KUKA KRL program: ps_ltc_res_c2.src, ps_ltc_res_c2.dat

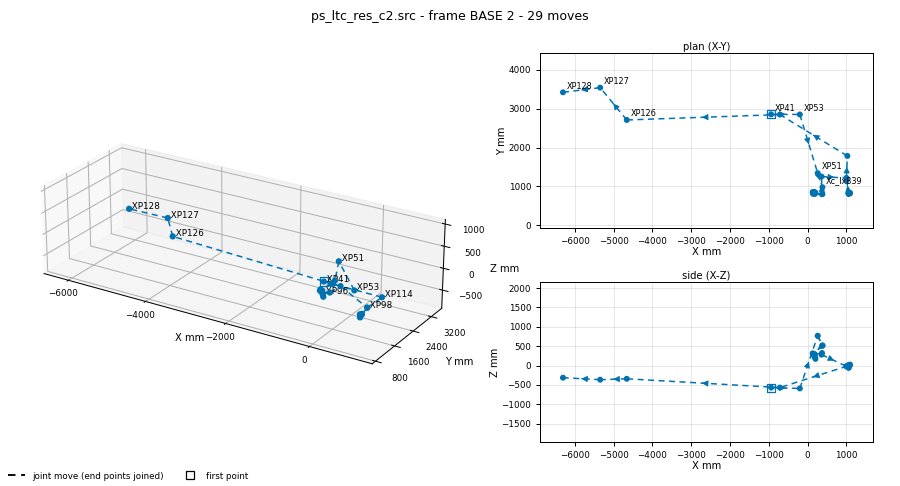
[picture p0: tool path of ps_ltc_res_c2.src in frame BASE 2, 29 of 30 moves have a stored position in this frame; points joined in program order, loops and branches not executed]
--- ps_ltc_res_c2.src ---
&ACCESS RVO2
&REL 51
&COMMENT Solda GUN C2 Respot
&PARAM DISKPATH = KRC:\R1\Program
DEF ps_ltc_res_c2( )
;FOLD INI
;FOLD SPOTTECH INI
USERSPOT(#INIT)
;ENDFOLD (SPOTTECH INI)
  ;FOLD USER INI
    ;Make your modifications here

  ;ENDFOLD (USER INI)
;ENDFOLD (INI)

; Caracterização dos meios de produção:
; Versão Atual:
; 15/07/2013 12:00 Name: P13.050-R4 CHANGES: Respot Acelo
; Pinça C2

chk_w2_wechs_ok ( )     ; CHECK FERRAMENTA: C2

;FOLD PTP P41 CONT Vel=100 % PDAT36 Tool[2]:GUN C2 Base[2]:ACCELO;%{PE}%R 8.2.20,%MKUKATPBASIS,%CMOVE,%VPTP,%P 1:PTP, 2:P41, 3:C_DIS, 5:100, 7:PDAT36
$BWDSTART=FALSE
PDAT_ACT=PPDAT36
FDAT_ACT=FP41
BAS(#PTP_PARAMS,100)
PTP XP41 C_DIS
;ENDFOLD

;FOLD OUT 3334 'R4 liberacao para solda respot' State=TRUE ;%{PE}%R 8.2.20,%MKUKATPBASIS,%COUT,%VOUTX,%P 2:3334, 3:R4 liberacao para solda respot, 5:TRUE, 6:
$OUT[3334]=TRUE
;ENDFOLD
;FOLD WAIT FOR ( IN 3334 'Aguarda lib soldar respot' );%{PE}%R 8.2.20,%MKUKATPBASIS,%CEXT_WAIT_FOR,%VEXT_WAIT_FOR,%P 2:, 4:, 5:$IN, 6:3334, 7:Aguarda lib soldar respot, 9:
WAIT FOR  ( $IN[3334] )
;ENDFOLD
;FOLD OUT 3334 'R4 solda respot concluida' State=FALSE ;%{PE}%R 8.2.20,%MKUKATPBASIS,%COUT,%VOUTX,%P 2:3334, 3:R4 solda respot concluida, 5:FALSE, 6:
$OUT[3334]=FALSE
;ENDFOLD
;FOLD OUT 3348 'Fora area GEOBOX' State=FALSE ;%{PE}%R 8.2.20,%MKUKATPBASIS,%COUT,%VOUTX,%P 2:3348, 3:Fora area GEOBOX, 5:FALSE, 6:
$OUT[3348]=FALSE
;ENDFOLD

;FOLD PTP P53 CONT Vel=100 % PDAT53 Tool[2]:GUN C2 Base[2]:ACCELO;%{PE}%R 8.2.20,%MKUKATPBASIS,%CMOVE,%VPTP,%P 1:PTP, 2:P53, 3:C_DIS, 5:100, 7:PDAT53
$BWDSTART=FALSE
PDAT_ACT=PPDAT53
FDAT_ACT=FP53
BAS(#PTP_PARAMS,100)
PTP XP53 C_DIS
;ENDFOLD
;FOLD PTP P51 CONT Vel=100 % PDAT51 Tool[2]:GUN C2 Base[2]:ACCELO;%{PE}%R 8.2.20,%MKUKATPBASIS,%CMOVE,%VPTP,%P 1:PTP, 2:P51, 3:C_DIS, 5:100, 7:PDAT51
$BWDSTART=FALSE
PDAT_ACT=PPDAT51
FDAT_ACT=FP51
BAS(#PTP_PARAMS,100)
PTP XP51 C_DIS
;ENDFOLD
;FOLD PTP c_lx839 CONT Vel=100 % P_OLP118 Tool[2]:GUN C2 Base[2]:ACCELO;%{PE}%R 8.2.20,%MKUKATPBASIS,%CMOVE,%VPTP,%P 1:PTP, 2:c_lx839, 3:C_DIS, 5:100, 7:P_OLP118
$BWDSTART=FALSE
PDAT_ACT=PP_OLP118
FDAT_ACT=Fc_lx839
BAS(#PTP_PARAMS,100)
PTP Xc_lx839 C_DIS
;ENDFOLD
;FOLD PTP P95 CONT Vel=100 % PDAT110 Tool[2]:GUN C2 Base[2]:ACCELO;%{PE}%R 8.2.20,%MKUKATPBASIS,%CMOVE,%VPTP,%P 1:PTP, 2:P95, 3:C_DIS, 5:100, 7:PDAT110
$BWDSTART=FALSE
PDAT_ACT=PPDAT110
FDAT_ACT=FP95
BAS(#PTP_PARAMS,100)
PTP XP95 C_DIS
;ENDFOLD
;FOLD PTP c_lx840 CONT Vel=100 % P_OLP119 Tool[2]:GUN C2 Base[2]:ACCELO;%{PE}%R 8.2.20,%MKUKATPBASIS,%CMOVE,%VPTP,%P 1:PTP, 2:c_lx840, 3:C_DIS, 5:100, 7:P_OLP119
$BWDSTART=FALSE
PDAT_ACT=PP_OLP119
FDAT_ACT=Fc_lx840
BAS(#PTP_PARAMS,100)
PTP Xc_lx840 C_DIS
;ENDFOLD

;FOLD ; swp_60_0224;%{PE}%R 8.2.20,%MKUKATPBASIS,%CCOMMENT,%VNORMAL,%P 2:swp_60_0224
;ENDFOLD
;FOLD PTP swp_60_0224 P_OLP120 SPOT Gun=2 RETR CLS PGNO1=106 ACTIVE=1 Tool[2]:GUN C2 Base[2]:ACCELO;%{PE}%R 8.2.2,%MKUKATPSPOT,%CSPOT,%VPTP,%P 1:PTP, 2:swp_60_0224, 3:, 5:100, 7:P_OLP120, 10:2, 12:#FIRST, 14:#CLO, 16:147, 18:1, 20:1, 22:0, 24:1, 25:S_OLP6
$BWDSTART=FALSE
PDAT_ACT=PP_OLP120
FDAT_ACT=Fswp_60_0224
BAS(#PTP_PARAMS,PP_OLP120.VEL)
S_ACT.GUN=2
S_ACT.PAIR=SDEFAULT.PAIR
S_ACT.RETR=#CLO
S_ACT.CLO_TM=1
S_ACT.PGNO1=106
S_ACT.PGNO2=SDEFAULT.PGNO2
S_ACT.PRESS1=SDEFAULT.PRESS1
S_ACT.PRESS2=SDEFAULT.PRESS2
S_READY=FALSE
PTP Xswp_60_0224
USERSPOT(#SPOT, S_ACT)
WAIT FOR S_READY
;ENDFOLD

;FOLD PTP c_lx841 CONT Vel=100 % P_OLP121 Tool[2]:GUN C2 Base[0];%{PE}%R 8.2.20,%MKUKATPBASIS,%CMOVE,%VPTP,%P 1:PTP, 2:c_lx841, 3:C_DIS, 5:100, 7:P_OLP121
$BWDSTART=FALSE
PDAT_ACT=PP_OLP121
FDAT_ACT=Fc_lx841
BAS(#PTP_PARAMS,100)
PTP Xc_lx841 C_DIS
;ENDFOLD

;FOLD ; swp_60_0228;%{PE}%R 8.2.20,%MKUKATPBASIS,%CCOMMENT,%VNORMAL,%P 2:swp_60_0228
;ENDFOLD
;FOLD PTP swp_60_0228 P_OLP122 SPOT Gun=2 RETR CLS PGNO1=138 ACTIVE=1 Tool[2]:GUN C2 Base[2]:ACCELO;%{PE}%R 8.2.2,%MKUKATPSPOT,%CSPOT,%VPTP,%P 1:PTP, 2:swp_60_0228, 3:, 5:100, 7:P_OLP122, 10:2, 12:#FIRST, 14:#CLO, 16:179, 18:1, 20:1, 22:0, 24:1, 25:S_OLP7
$BWDSTART=FALSE
PDAT_ACT=PP_OLP122
FDAT_ACT=Fswp_60_0228
BAS(#PTP_PARAMS,PP_OLP122.VEL)
S_ACT.GUN=2
S_ACT.PAIR=SDEFAULT.PAIR
S_ACT.RETR=#CLO
S_ACT.CLO_TM=1
S_ACT.PGNO1=138
S_ACT.PGNO2=SDEFAULT.PGNO2
S_ACT.PRESS1=SDEFAULT.PRESS1
S_ACT.PRESS2=SDEFAULT.PRESS2
S_READY=FALSE
PTP Xswp_60_0228
USERSPOT(#SPOT, S_ACT)
WAIT FOR S_READY
;ENDFOLD

;FOLD ; swp_60_0232;%{PE}%R 8.2.20,%MKUKATPBASIS,%CCOMMENT,%VNORMAL,%P 2:swp_60_0232
;ENDFOLD
;FOLD PTP swp_60_0232 P_OLP123 SPOT Gun=2 RETR CLS PGNO1=104 ACTIVE=1 Tool[2]:GUN C2 Base[2]:ACCELO;%{PE}%R 8.2.2,%MKUKATPSPOT,%CSPOT,%VPTP,%P 1:PTP, 2:swp_60_0232, 3:, 5:100, 7:P_OLP123, 10:2, 12:#FIRST, 14:#CLO, 16:145, 18:1, 20:1, 22:0, 24:1, 25:S_OLP8
$BWDSTART=FALSE
PDAT_ACT=PP_OLP123
FDAT_ACT=Fswp_60_0232
BAS(#PTP_PARAMS,PP_OLP123.VEL)
S_ACT.GUN=2
S_ACT.PAIR=SDEFAULT.PAIR
S_ACT.RETR=#CLO
S_ACT.CLO_TM=1
S_ACT.PGNO1=104
S_ACT.PGNO2=SDEFAULT.PGNO2
S_ACT.PRESS1=SDEFAULT.PRESS1
S_ACT.PRESS2=SDEFAULT.PRESS2
S_READY=FALSE
PTP Xswp_60_0232
USERSPOT(#SPOT, S_ACT)
WAIT FOR S_READY
;ENDFOLD

;FOLD PTP P96 CONT Vel=100 % PDAT111 Tool[2]:GUN C2 Base[2]:ACCELO;%{PE}%R 8.2.20,%MKUKATPBASIS,%CMOVE,%VPTP,%P 1:PTP, 2:P96, 3:C_DIS, 5:100, 7:PDAT111
$BWDSTART=FALSE
PDAT_ACT=PPDAT111
FDAT_ACT=FP96
BAS(#PTP_PARAMS,100)
PTP XP96 C_DIS
;ENDFOLD

;FOLD ; swp_60_0234;%{PE}%R 8.2.20,%MKUKATPBASIS,%CCOMMENT,%VNORMAL,%P 2:swp_60_0234
;ENDFOLD
;FOLD PTP swp_60_0234 PDAT112 SPOT Gun=2 RETR OPN PGNO1=103 ACTIVE=1 Tool[2]:GUN C2 Base[2]:ACCELO;%{PE}%R 8.2.2,%MKUKATPSPOT,%CSPOT,%VPTP,%P 1:PTP, 2:swp_60_0234, 3:, 5:100, 7:PDAT112, 10:2, 12:#FIRST, 14:#OPN, 16:144, 18:1, 20:0, 22:0, 24:1, 25:NORMAL
$BWDSTART=FALSE
PDAT_ACT=PPDAT112
FDAT_ACT=Fswp_60_0234
BAS(#PTP_PARAMS,PPDAT112.VEL)
S_ACT.GUN=2
S_ACT.PAIR=SDEFAULT.PAIR
S_ACT.RETR=#OPN
S_ACT.CLO_TM=1
S_ACT.PGNO1=103
S_ACT.PGNO2=SDEFAULT.PGNO2
S_ACT.PRESS1=SDEFAULT.PRESS1
S_ACT.PRESS2=SDEFAULT.PRESS2
S_READY=FALSE
PTP Xswp_60_0234
USERSPOT(#SPOT, S_ACT)
WAIT FOR S_READY
;ENDFOLD

;FOLD PTP c_lx804 CONT Vel=100 % P_OLP124 Tool[2]:GUN C2 Base[2]:ACCELO;%{PE}%R 8.2.20,%MKUKATPBASIS,%CMOVE,%VPTP,%P 1:PTP, 2:c_lx804, 3:C_DIS, 5:100, 7:P_OLP124
$BWDSTART=FALSE
PDAT_ACT=PP_OLP124
FDAT_ACT=Fc_lx804
BAS(#PTP_PARAMS,100)
PTP Xc_lx804 C_DIS
;ENDFOLD
;FOLD PTP P94 CONT Vel=100 % PDAT109 Tool[2]:GUN C2 Base[2]:ACCELO;%{PE}%R 8.2.20,%MKUKATPBASIS,%CMOVE,%VPTP,%P 1:PTP, 2:P94, 3:C_DIS, 5:100, 7:PDAT109
$BWDSTART=FALSE
PDAT_ACT=PPDAT109
FDAT_ACT=FP94
BAS(#PTP_PARAMS,100)
PTP XP94 C_DIS
;ENDFOLD
;FOLD PTP c_lx807 Vel=100 % P_OLP125 Tool[2]:GUN C2 Base[2]:ACCELO;%{PE}%R 8.2.20,%MKUKATPBASIS,%CMOVE,%VPTP,%P 1:PTP, 2:c_lx807, 3:, 5:100, 7:P_OLP125
$BWDSTART=FALSE
PDAT_ACT=PP_OLP125
FDAT_ACT=Fc_lx807
BAS(#PTP_PARAMS,100)
PTP Xc_lx807
;ENDFOLD

;FOLD Collision.Monitoring_AREA_1_On ;%{PE}%MKUKATPUSER
COLLSTOP( 7, 1 ) ;not Interrupt-Controlled
;ENDFOLD

;FOLD PTP P98 CONT Vel=100 % PDAT114 Tool[2]:GUN C2 Base[2]:ACCELO;%{PE}%R 8.2.20,%MKUKATPBASIS,%CMOVE,%VPTP,%P 1:PTP, 2:P98, 3:C_DIS, 5:100, 7:PDAT114
$BWDSTART=FALSE
PDAT_ACT=PPDAT114
FDAT_ACT=FP98
BAS(#PTP_PARAMS,100)
PTP XP98 C_DIS
;ENDFOLD
;FOLD PTP P99 CONT Vel=100 % PDAT115 Tool[2]:GUN C2 Base[2]:ACCELO;%{PE}%R 8.2.20,%MKUKATPBASIS,%CMOVE,%VPTP,%P 1:PTP, 2:P99, 3:C_DIS, 5:100, 7:PDAT115
$BWDSTART=FALSE
PDAT_ACT=PPDAT115
FDAT_ACT=FP99
BAS(#PTP_PARAMS,100)
PTP XP99 C_DIS
;ENDFOLD
;FOLD PTP P100 CONT Vel=100 % PDAT116 Tool[2]:GUN C2 Base[2]:ACCELO;%{PE}%R 8.2.20,%MKUKATPBASIS,%CMOVE,%VPTP,%P 1:PTP, 2:P100, 3:C_DIS, 5:100, 7:PDAT116
$BWDSTART=FALSE
PDAT_ACT=PPDAT116
FDAT_ACT=FP100
BAS(#PTP_PARAMS,100)
PTP XP100 C_DIS
;ENDFOLD
;FOLD PTP P101 CONT Vel=100 % PDAT118 Tool[2]:GUN C2 Base[2]:ACCELO;%{PE}%R 8.2.20,%MKUKATPBASIS,%CMOVE,%VPTP,%P 1:PTP, 2:P101, 3:C_DIS, 5:100, 7:PDAT118
$BWDSTART=FALSE
PDAT_ACT=PPDAT118
FDAT_ACT=FP101
BAS(#PTP_PARAMS,100)
PTP XP101 C_DIS
;ENDFOLD

;FOLD ; 60_0310;%{PE}%R 8.2.20,%MKUKATPBASIS,%CCOMMENT,%VNORMAL,%P 2:60_0310
;ENDFOLD
;FOLD PTP swp_60_0310 PDAT128 SPOT Gun=2 RETR CLS PGNO1=85 ACTIVE=1 Tool[2]:GUN C2 Base[2]:ACCELO;%{PE}%R 8.2.2,%MKUKATPSPOT,%CSPOT,%VPTP,%P 1:PTP, 2:swp_60_0310, 3:, 5:100, 7:PDAT128, 10:2, 12:#FIRST, 14:#CLO, 16:126, 18:1, 20:0, 22:0, 24:1, 25:NORMAL
$BWDSTART=FALSE
PDAT_ACT=PPDAT128
FDAT_ACT=Fswp_60_0310
BAS(#PTP_PARAMS,PPDAT128.VEL)
S_ACT.GUN=2
S_ACT.PAIR=SDEFAULT.PAIR
S_ACT.RETR=#CLO
S_ACT.CLO_TM=1
S_ACT.PGNO1=85
S_ACT.PGNO2=SDEFAULT.PGNO2
S_ACT.PRESS1=SDEFAULT.PRESS1
S_ACT.PRESS2=SDEFAULT.PRESS2
S_READY=FALSE
PTP Xswp_60_0310
USERSPOT(#SPOT, S_ACT)
WAIT FOR S_READY
;ENDFOLD

;FOLD ; 60_0308;%{PE}%R 8.2.20,%MKUKATPBASIS,%CCOMMENT,%VNORMAL,%P 2:60_0308
;ENDFOLD
;FOLD PTP swp_60_0308 PDAT129 SPOT Gun=2 RETR OPN PGNO1=139 ACTIVE=1 Tool[2]:GUN C2 Base[2]:ACCELO;%{PE}%R 8.2.2,%MKUKATPSPOT,%CSPOT,%VPTP,%P 1:PTP, 2:swp_60_0308, 3:, 5:100, 7:PDAT129, 10:2, 12:#FIRST, 14:#OPN, 16:180, 18:1, 20:0, 22:0, 24:1, 25:NORMAL
$BWDSTART=FALSE
PDAT_ACT=PPDAT129
FDAT_ACT=Fswp_60_0308
BAS(#PTP_PARAMS,PPDAT129.VEL)
S_ACT.GUN=2
S_ACT.PAIR=SDEFAULT.PAIR
S_ACT.RETR=#OPN
S_ACT.CLO_TM=1
S_ACT.PGNO1=139
S_ACT.PGNO2=SDEFAULT.PGNO2
S_ACT.PRESS1=SDEFAULT.PRESS1
S_ACT.PRESS2=SDEFAULT.PRESS2
S_READY=FALSE
PTP Xswp_60_0308
USERSPOT(#SPOT, S_ACT)
WAIT FOR S_READY
;ENDFOLD

;FOLD PTP P110 CONT Vel=100 % PDAT130 Tool[2]:GUN C2 Base[2]:ACCELO;%{PE}%R 8.2.20,%MKUKATPBASIS,%CMOVE,%VPTP,%P 1:PTP, 2:P110, 3:C_DIS, 5:100, 7:PDAT130
$BWDSTART=FALSE
PDAT_ACT=PPDAT130
FDAT_ACT=FP110
BAS(#PTP_PARAMS,100)
PTP XP110 C_DIS
;ENDFOLD
;FOLD PTP P111 CONT Vel=100 % PDAT131 Tool[2]:GUN C2 Base[2]:ACCELO;%{PE}%R 8.2.20,%MKUKATPBASIS,%CMOVE,%VPTP,%P 1:PTP, 2:P111, 3:C_DIS, 5:100, 7:PDAT131
$BWDSTART=FALSE
PDAT_ACT=PPDAT131
FDAT_ACT=FP111
BAS(#PTP_PARAMS,100)
PTP XP111 C_DIS
;ENDFOLD
;FOLD PTP P112 CONT Vel=100 % PDAT132 Tool[2]:GUN C2 Base[2]:ACCELO;%{PE}%R 8.2.20,%MKUKATPBASIS,%CMOVE,%VPTP,%P 1:PTP, 2:P112, 3:C_DIS, 5:100, 7:PDAT132
$BWDSTART=FALSE
PDAT_ACT=PPDAT132
FDAT_ACT=FP112
BAS(#PTP_PARAMS,100)
PTP XP112 C_DIS
;ENDFOLD
;FOLD PTP P114 CONT Vel=100 % PDAT134 Tool[2]:GUN C2 Base[2]:ACCELO;%{PE}%R 8.2.20,%MKUKATPBASIS,%CMOVE,%VPTP,%P 1:PTP, 2:P114, 3:C_DIS, 5:100, 7:PDAT134
$BWDSTART=FALSE
PDAT_ACT=PPDAT134
FDAT_ACT=FP114
BAS(#PTP_PARAMS,100)
PTP XP114 C_DIS
;ENDFOLD
;FOLD PTP P109 CONT Vel=100 % PDAT127 Tool[2]:GUN C2 Base[2]:ACCELO;%{PE}%R 8.2.20,%MKUKATPBASIS,%CMOVE,%VPTP,%P 1:PTP, 2:P109, 3:C_DIS, 5:100, 7:PDAT127
$BWDSTART=FALSE
PDAT_ACT=PPDAT127
FDAT_ACT=FP109
BAS(#PTP_PARAMS,100)
PTP XP109 C_DIS
;ENDFOLD
;FOLD PTP P126 CONT Vel=100 % PDAT146 Tool[2]:GUN C2 Base[2]:ACCELO;%{PE}%R 8.2.20,%MKUKATPBASIS,%CMOVE,%VPTP,%P 1:PTP, 2:P126, 3:C_DIS, 5:100, 7:PDAT146
$BWDSTART=FALSE
PDAT_ACT=PPDAT146
FDAT_ACT=FP126
BAS(#PTP_PARAMS,100)
PTP XP126 C_DIS
;ENDFOLD
;FOLD PTP P127 CONT Vel=100 % PDAT147 Tool[2]:GUN C2 Base[2]:ACCELO;%{PE}%R 8.2.20,%MKUKATPBASIS,%CMOVE,%VPTP,%P 1:PTP, 2:P127, 3:C_DIS, 5:100, 7:PDAT147
$BWDSTART=FALSE
PDAT_ACT=PPDAT147
FDAT_ACT=FP127
BAS(#PTP_PARAMS,100)
PTP XP127 C_DIS
;ENDFOLD
;FOLD PTP P128 CONT Vel=100 % PDAT148 Tool[2]:GUN C2 Base[2]:ACCELO;%{PE}%R 8.2.20,%MKUKATPBASIS,%CMOVE,%VPTP,%P 1:PTP, 2:P128, 3:C_DIS, 5:100, 7:PDAT148
$BWDSTART=FALSE
PDAT_ACT=PPDAT148
FDAT_ACT=FP128
BAS(#PTP_PARAMS,100)
PTP XP128 C_DIS
;ENDFOLD

;FOLD PULSE 3345 'Solda Respot concluida' State=TRUE Time=1 sec;%{PE}%R 8.2.20,%MKUKATPBASIS,%COUT,%VPULSE,%P 2:3345, 3:Solda Respot concluida, 5:TRUE, 6:, 8:1
PULSE($OUT[3345], TRUE,1)
;ENDFOLD
;FOLD OUT 3348 'Fora area GEOBOX' State=TRUE ;%{PE}%R 8.2.20,%MKUKATPBASIS,%COUT,%VOUTX,%P 2:3348, 3:Fora area GEOBOX, 5:TRUE, 6:
$OUT[3348]=TRUE
;ENDFOLD
;FOLD Collision.Monitoring_AREA_1_Off . ;%{PE}%MKUKATPUSER
COLLSTOP( 7, 2+0 )
;ENDFOLD

;FOLD PTP P121 Vel=100 % PDAT141 Tool[2]:GUN C2 Base[0];%{PE}%R 8.2.20,%MKUKATPBASIS,%CMOVE,%VPTP,%P 1:PTP, 2:P121, 3:, 5:100, 7:PDAT141
$BWDSTART=FALSE
PDAT_ACT=PPDAT141
FDAT_ACT=FP121
BAS(#PTP_PARAMS,100)
PTP XP121
;ENDFOLD

if FraesAnf (2) then
  f_fraes2 ()
endif

END

--- ps_ltc_res_c2.dat ---
&ACCESS RVO2
&REL 51
&COMMENT Solda GUN C2 Respot
&PARAM DISKPATH = KRC:\R1\Program
DEFDAT  ps_ltc_res_c2
;FOLD EXTERNAL DECLARATIONS;%{PE}%MKUKATPBASIS,%CEXT,%VCOMMON,%P
;FOLD GRIPPERTECH EXT
EXT  H50 (INT  :IN,INT  :IN,INT  :IN,GRP_TYP  :IN )
;ENDFOLD (GRIPPERTECH EXT)
;FOLD SPOTTECH EXT
EXT  USERSPOT (S_COMMAND  :IN,SPOT_TYPE  :IN )
;ENDFOLD (SPOTTECH EXT)
;FOLD BASISTECH EXT;%{PE}%MKUKATPBASIS,%CEXT,%VEXT,%P
EXT  BAS (BAS_COMMAND  :IN,REAL  :IN )
DECL INT SUCCESS
;ENDFOLD (BASISTECH EXT)
;FOLD USER EXT;%{E}%MKUKATPUSER,%CEXT,%VEXT,%P
;Make your modifications here

;ENDFOLD (USER EXT)
;ENDFOLD (EXTERNAL DECLARATIONS)

;# ============ START PATH : swp_p13050r4_ltc_res_c2 =============
DECL SPOT_TYPE SS_OLP1={GUN 1,PAIR #FIRST,RETR #OPN,CLO_TM 0,PGNO1 1,PRESS1 1.0,PGNO2 0,PRESS2 0.0}
DECL SPOT_TYPE SS_OLP2={GUN 1,PAIR #FIRST,RETR #OPN,CLO_TM 0,PGNO1 1,PRESS1 1.0,PGNO2 0,PRESS2 0.0}
DECL SPOT_TYPE SS_OLP3={GUN 1,PAIR #FIRST,RETR #OPN,CLO_TM 0,PGNO1 1,PRESS1 1.0,PGNO2 0,PRESS2 0.0}
DECL SPOT_TYPE SS_OLP4={GUN 1,PAIR #FIRST,RETR #OPN,CLO_TM 0,PGNO1 1,PRESS1 1.0,PGNO2 0,PRESS2 0.0}
DECL SPOT_TYPE SS_OLP5={GUN 1,PAIR #FIRST,RETR #OPN,CLO_TM 0,PGNO1 1,PRESS1 1.0,PGNO2 0,PRESS2 0.0}
DECL SPOT_TYPE SS_OLP6={GUN 1,PAIR #FIRST,RETR #OPN,CLO_TM 0,PGNO1 1,PRESS1 1.0,PGNO2 0,PRESS2 0.0}
DECL SPOT_TYPE SS_OLP7={GUN 1,PAIR #FIRST,RETR #OPN,CLO_TM 0,PGNO1 1,PRESS1 1.0,PGNO2 0,PRESS2 0.0}
DECL FDAT Fswp_60_0308={TOOL_NO 2,BASE_NO 2,IPO_FRAME #BASE,POINT2[] " "}
DECL SPOT_TYPE SS_OLP8={GUN 1,PAIR #FIRST,RETR #OPN,CLO_TM 0,PGNO1 1,PRESS1 1.0,PGNO2 0,PRESS2 0.0}
DECL E6POS Xswp_60_0308={X 1096.53198,Y 822.993225,Z 14.3700304,A 1.80438006,B -53.1394386,C -88.516777,S 2,T 2,E1 5392.10791,E2 0.0,E3 0.0,E4 0.0,E5 0.0,E6 0.0}
DECL FDAT Fswp_60_0310={TOOL_NO 2,BASE_NO 2,IPO_FRAME #BASE,POINT2[] " "}
DECL SPOT_TYPE SS_OLP9={GUN 1,PAIR #FIRST,RETR #OPN,CLO_TM 0,PGNO1 1,PRESS1 1.0,PGNO2 0,PRESS2 0.0}
DECL E6POS Xswp_60_0310={X 1094.51404,Y 825.377197,Z 26.2432995,A 1.79304504,B -53.1312599,C -88.5010376,S 2,T 2,E1 5392.10889,E2 0.0,E3 0.0,E4 0.0,E5 0.0,E6 0.0}
DECL SPOT_TYPE SS_OLP10={GUN 1,PAIR #FIRST,RETR #OPN,CLO_TM 0,PGNO1 1,PRESS1 1.0,PGNO2 0,PRESS2 0.0}
DECL SPOT_TYPE SS_OLP11={GUN 1,PAIR #FIRST,RETR #OPN,CLO_TM 0,PGNO1 1,PRESS1 1.0,PGNO2 0,PRESS2 0.0}
DECL SPOT_TYPE SS_OLP12={GUN 1,PAIR #FIRST,RETR #OPN,CLO_TM 0,PGNO1 1,PRESS1 1.0,PGNO2 0,PRESS2 0.0}
DECL SPOT_TYPE SS_OLP13={GUN 1,PAIR #FIRST,RETR #OPN,CLO_TM 0,PGNO1 1,PRESS1 1.0,PGNO2 0,PRESS2 0.0}
DECL SPOT_TYPE SS_OLP14={GUN 1,PAIR #FIRST,RETR #OPN,CLO_TM 0,PGNO1 1,PRESS1 1.0,PGNO2 0,PRESS2 0.0}
DECL SPOT_TYPE SS_OLP15={GUN 1,PAIR #FIRST,RETR #OPN,CLO_TM 0,PGNO1 1,PRESS1 1.0,PGNO2 0,PRESS2 0.0}
DECL SPOT_TYPE SS_OLP16={GUN 1,PAIR #FIRST,RETR #OPN,CLO_TM 0,PGNO1 1,PRESS1 1.0,PGNO2 0,PRESS2 0.0}
DECL SPOT_TYPE SS_OLP17={GUN 1,PAIR #FIRST,RETR #OPN,CLO_TM 0,PGNO1 1,PRESS1 1.0,PGNO2 0,PRESS2 0.0}
DECL SPOT_TYPE SS_OLP18={GUN 1,PAIR #FIRST,RETR #OPN,CLO_TM 0,PGNO1 1,PRESS1 1.0,PGNO2 0,PRESS2 0.0}
DECL SPOT_TYPE SS_OLP19={GUN 1,PAIR #FIRST,RETR #OPN,CLO_TM 0,PGNO1 1,PRESS1 1.0,PGNO2 0,PRESS2 0.0}
DECL SPOT_TYPE SS_OLP20={GUN 1,PAIR #FIRST,RETR #OPN,CLO_TM 0,PGNO1 1,PRESS1 1.0,PGNO2 0,PRESS2 0.0}
DECL SPOT_TYPE SS_OLP21={GUN 1,PAIR #FIRST,RETR #OPN,CLO_TM 0,PGNO1 1,PRESS1 1.0,PGNO2 0,PRESS2 0.0}
DECL SPOT_TYPE SS_OLP22={GUN 1,PAIR #FIRST,RETR #OPN,CLO_TM 0,PGNO1 1,PRESS1 1.0,PGNO2 0,PRESS2 0.0}
DECL SPOT_TYPE SS_OLP23={GUN 1,PAIR #FIRST,RETR #OPN,CLO_TM 0,PGNO1 1,PRESS1 1.0,PGNO2 0,PRESS2 0.0}
DECL SPOT_TYPE SS_OLP24={GUN 1,PAIR #FIRST,RETR #OPN,CLO_TM 0,PGNO1 1,PRESS1 1.0,PGNO2 0,PRESS2 0.0}
DECL FDAT Fswp_60_0234={TOOL_NO 2,BASE_NO 2,IPO_FRAME #BASE,POINT2[] " "}
DECL SPOT_TYPE SS_OLP25={GUN 1,PAIR #FIRST,RETR #OPN,CLO_TM 0,PGNO1 1,PRESS1 1.0,PGNO2 0,PRESS2 0.0}
DECL E6POS Xswp_60_0234={X 205.289398,Y 834.686523,Z 173.667694,A 176.962494,B 30.1434307,C 87.1450806,S 2,T 34,E1 5342.354,E2 0.0,E3 0.0,E4 0.0,E5 0.0,E6 0.0}
DECL FDAT Fswp_60_0232={TOOL_NO 2,BASE_NO 2,IPO_FRAME #BASE,POINT2[] " "}
DECL SPOT_TYPE SS_OLP26={GUN 1,PAIR #FIRST,RETR #OPN,CLO_TM 0,PGNO1 1,PRESS1 1.0,PGNO2 0,PRESS2 0.0}
DECL E6POS Xswp_60_0232={X 179.287292,Y 847.949585,Z 228.299698,A 179.160507,B 20.9243603,C 87.9932938,S 2,T 34,E1 5342.33203,E2 0.0,E3 0.0,E4 0.0,E5 0.0,E6 0.0}
DECL FDAT Fswp_60_0228={TOOL_NO 2,BASE_NO 2,IPO_FRAME #BASE,POINT2[] " "}
DECL SPOT_TYPE SS_OLP27={GUN 1,PAIR #FIRST,RETR #OPN,CLO_TM 0,PGNO1 1,PRESS1 1.0,PGNO2 0,PRESS2 0.0}
DECL E6POS Xswp_60_0228={X 166.7827,Y 849.044617,Z 275.148712,A 175.758102,B 30.2118301,C 88.6927338,S 2,T 34,E1 5342.34277,E2 0.0,E3 0.0,E4 0.0,E5 0.0,E6 0.0}
DECL FDAT Fswp_60_0224={TOOL_NO 2,BASE_NO 2,IPO_FRAME #BASE,POINT2[] " "}
DECL SPOT_TYPE SS_OLP28={GUN 1,PAIR #FIRST,RETR #OPN,CLO_TM 0,PGNO1 1,PRESS1 1.0,PGNO2 0,PRESS2 0.0}
DECL E6POS Xswp_60_0224={X 132.417099,Y 851.122925,Z 315.260712,A 176.934692,B 7.25355816,C 88.1791992,S 2,T 34,E1 5341.85986,E2 0.0,E3 0.0,E4 0.0,E5 0.0,E6 0.0}
DECL SPOT_TYPE SS_OLP29={GUN 1,PAIR #FIRST,RETR #OPN,CLO_TM 0,PGNO1 1,PRESS1 1.0,PGNO2 0,PRESS2 0.0}
DECL SPOT_TYPE SS_OLP30={GUN 1,PAIR #FIRST,RETR #OPN,CLO_TM 0,PGNO1 1,PRESS1 1.0,PGNO2 0,PRESS2 0.0}
DECL SPOT_TYPE SS_OLP31={GUN 1,PAIR #FIRST,RETR #OPN,CLO_TM 0,PGNO1 1,PRESS1 1.0,PGNO2 0,PRESS2 0.0}
DECL BASIS_SUGG_T LAST_BASIS={POINT1[] "P128                    ",POINT2[] "P128                    ",CP_PARAMS[] "CPDAT0                  ",PTP_PARAMS[] "PDAT148                 ",CONT[] "C_DIS                   ",CP_VEL[] "2.0                     ",PTP_VEL[] "100                     ",SYNC_PARAMS[] "SYNCDAT                 ",SPL_NAME[] "S0                      "}
DECL SPOT_SUGG_T LAST_SPOT={GUN[] "2                       ",RETR_CMD[] "#OPN                    ",CHOISE[] "#FIRST                  ",CLO_TM[] "1                       ",PGNO1[] "159                     ",PRESS1[] "0                       ",PGNO2[] "1                       ",PRESS2[] "0                       ",SPOT_PARAMS[] "NORMAL                  "}
DECL PDAT PPDAT36={VEL 100.0,ACC 100.0,APO_DIST 100.0,APO_MODE #CDIS}
DECL E6POS XP41={X -937.438416,Y 2856.41602,Z -568.258484,A 111.187798,B -1.17266095,C -11.4579496,S 2,T 42,E1 4076.13306,E2 0.0,E3 0.0,E4 0.0,E5 0.0,E6 0.0}
DECL FDAT FP41={TOOL_NO 1,BASE_NO 2,IPO_FRAME #BASE,POINT2[] " ",TQ_STATE FALSE}
DECL PDAT PPDAT51={VEL 100.0,ACC 100.0,APO_DIST 100.0,APO_MODE #CDIS}
DECL E6POS XP51={X 262.233093,Y 1339.60303,Z 770.668884,A -164.779205,B 56.1851616,C 83.1335907,S 2,T 34,E1 5014.16992,E2 0.0,E3 0.0,E4 0.0,E5 0.0,E6 0.0}
DECL FDAT FP51={TOOL_NO 1,BASE_NO 2,IPO_FRAME #BASE,POINT2[] " ",TQ_STATE FALSE}
DECL PDAT PPDAT53={VEL 100.0,ACC 100.0,APO_DIST 100.0,APO_MODE #CDIS}
DECL E6POS XP53={X -197.839706,Y 2852.4541,Z -588.636414,A 111.435501,B -4.20538092,C -4.20640898,S 2,T 42,E1 5014.16992,E2 0.0,E3 0.0,E4 0.0,E5 0.0,E6 0.0}
DECL FDAT FP53={TOOL_NO 2,BASE_NO 2,IPO_FRAME #BASE,POINT2[] " ",TQ_STATE FALSE}
DECL PDAT PP_OLP118={VEL 100.0,ACC 100.0,APO_DIST 100.0,APO_MODE #CDIS}
DECL E6POS Xc_lx839={X 384.908112,Y 975.687378,Z 517.934021,A -173.897995,B 25.5046997,C 87.3456268,S 2,T 34,E1 5216.62988,E2 0.0,E3 0.0,E4 0.0,E5 0.0,E6 0.0}
DECL FDAT Fc_lx839={TOOL_NO 2,BASE_NO 2,IPO_FRAME #BASE,POINT2[] " "}
DECL PDAT PP_OLP119={VEL 100.0,ACC 100.0,APO_DIST 100.0,APO_MODE #CDIS}
DECL E6POS Xc_lx840={X 141.115601,Y 807.457825,Z 303.338806,A 175.901703,B 18.8709393,C 88.7724228,S 2,T 34,E1 5341.79395,E2 0.0,E3 0.0,E4 0.0,E5 0.0,E6 0.0}
DECL FDAT Fc_lx840={TOOL_NO 2,BASE_NO 2,IPO_FRAME #BASE,POINT2[] " "}
DECL PDAT PP_OLP120={VEL 100.0,ACC 100.0,APO_DIST 0.0}
DECL PDAT PP_OLP121={VEL 100.0,ACC 100.0,APO_DIST 100.0,APO_MODE #CDIS}
DECL E6POS Xc_lx841={X 168.147202,Y 843.355713,Z 297.313385,A 175.906906,B 24.1678505,C 88.7748718,S 2,T 34,E1 5342.34424,E2 0.0,E3 0.0,E4 0.0,E5 0.0,E6 0.0}
DECL FDAT Fc_lx841={TOOL_NO 2,BASE_NO 2,IPO_FRAME #BASE,POINT2[] " "}
DECL PDAT PP_OLP122={VEL 100.0,ACC 100.0,APO_DIST 0.0}
DECL PDAT PP_OLP123={VEL 100.0,ACC 100.0,APO_DIST 0.0}
DECL PDAT PP_OLP124={VEL 100.0,ACC 100.0,APO_DIST 100.0,APO_MODE #CDIS}
DECL E6POS Xc_lx804={X 188.816101,Y 801.955383,Z 290.867401,A 175.750305,B 32.2371292,C 88.6945496,S 2,T 34,E1 5342.53711,E2 0.0,E3 0.0,E4 0.0,E5 0.0,E6 0.0}
DECL FDAT Fc_lx804={TOOL_NO 2,BASE_NO 2,IPO_FRAME #BASE,POINT2[] " "}
DECL PDAT PPDAT109={VEL 100.0,ACC 100.0,APO_DIST 100.0,APO_MODE #CDIS}
DECL E6POS XP94={X 373.632599,Y 795.344116,Z 324.714386,A -179.201599,B 45.2583389,C 88.5806732,S 2,T 34,E1 5364.28711,E2 0.0,E3 0.0,E4 0.0,E5 0.0,E6 0.0}
DECL FDAT FP94={TOOL_NO 2,BASE_NO 2,IPO_FRAME #BASE,POINT2[] " ",TQ_STATE FALSE}
DECL PDAT PP_OLP125={VEL 100.0,ACC 100.0,APO_DIST 100.0,APO_MODE #CDIS}
DECL E6POS Xc_lx807={X 361.210114,Y 1251.96399,Z 281.714294,A -172.720001,B 54.0112801,C 88.4402008,S 2,T 34,E1 5392.10205,E2 0.0,E3 0.0,E4 0.0,E5 0.0,E6 0.0}
DECL FDAT Fc_lx807={TOOL_NO 2,BASE_NO 2,IPO_FRAME #BASE,POINT2[] " "}
DECL E6POS XP95={X 385.754089,Y 801.401794,Z 517.934204,A -173.897903,B 25.5047894,C 87.3456726,S 2,T 34,E1 5216.62988,E2 0.0,E3 0.0,E4 0.0,E5 0.0,E6 0.0}
DECL FDAT FP95={TOOL_NO 2,BASE_NO 2,IPO_FRAME #BASE,POINT2[] " ",TQ_STATE FALSE}
DECL PDAT PPDAT110={VEL 100.0,ACC 100.0,APO_DIST 100.0,APO_MODE #CDIS}
DECL E6POS XP96={X 192.183304,Y 839.262695,Z 219.117096,A 176.966904,B 30.1538105,C 87.1508636,S 2,T 34,E1 5342.35596,E2 0.0,E3 0.0,E4 0.0,E5 0.0,E6 0.0}
DECL FDAT FP96={TOOL_NO 2,BASE_NO 2,IPO_FRAME #BASE,POINT2[] " ",TQ_STATE FALSE}
DECL PDAT PPDAT111={VEL 100.0,ACC 100.0,APO_DIST 100.0,APO_MODE #CDIS}
DECL PDAT PPDAT112={VEL 100.0,ACC 100.0,APO_DIST 100.0}
DECL E6POS XP98={X 1003.49402,Y 1211.99597,Z -19.1957207,A 6.74869108,B -43.3641891,C -92.4024506,S 2,T 2,E1 5392.104,E2 0.0,E3 0.0,E4 0.0,E5 0.0,E6 0.0}
DECL FDAT FP98={TOOL_NO 2,BASE_NO 2,IPO_FRAME #BASE,POINT2[] " ",TQ_STATE FALSE}
DECL PDAT PPDAT114={VEL 100.0,ACC 100.0,APO_DIST 100.0,APO_MODE #CDIS}
DECL E6POS XP99={X 1060.797,Y 818.631897,Z -47.6112289,A 6.91774082,B -40.6273918,C -92.0087128,S 2,T 2,E1 5392.104,E2 0.0,E3 0.0,E4 0.0,E5 0.0,E6 0.0}
DECL FDAT FP99={TOOL_NO 2,BASE_NO 2,IPO_FRAME #BASE,POINT2[] " ",TQ_STATE FALSE}
DECL PDAT PPDAT115={VEL 100.0,ACC 100.0,APO_DIST 100.0,APO_MODE #CDIS}
DECL E6POS XP100={X 1060.77698,Y 818.632385,Z -11.0750799,A 7.32021999,B -48.3009911,C -92.2918015,S 2,T 2,E1 5392.10498,E2 0.0,E3 0.0,E4 0.0,E5 0.0,E6 0.0}
DECL FDAT FP100={TOOL_NO 2,BASE_NO 2,IPO_FRAME #BASE,POINT2[] " ",TQ_STATE FALSE}
DECL PDAT PPDAT116={VEL 100.0,ACC 100.0,APO_DIST 100.0,APO_MODE #CDIS}
DECL E6POS XP101={X 1064.172,Y 802.139282,Z 16.5553303,A 7.57951689,B -52.4292908,C -92.4938736,S 2,T 2,E1 5392.10596,E2 0.0,E3 0.0,E4 0.0,E5 0.0,E6 0.0}
DECL FDAT FP101={TOOL_NO 2,BASE_NO 2,IPO_FRAME #BASE,POINT2[] " ",TQ_STATE FALSE}
DECL PDAT PPDAT118={VEL 100.0,ACC 100.0,APO_DIST 100.0,APO_MODE #CDIS}
DECL E6POS XP109={X -712.520508,Y 2849.75806,Z -566.928528,A 111.187897,B -1.17260897,C -11.4580898,S 2,T 42,E1 4298.78809,E2 0.0,E3 0.0,E4 0.0,E5 0.0,E6 0.0}
DECL FDAT FP109={TOOL_NO 2,BASE_NO 2,IPO_FRAME #BASE,POINT2[] " ",TQ_STATE FALSE}
DECL PDAT PPDAT127={VEL 100.0,ACC 100.0,APO_DIST 100.0,APO_MODE #CDIS}
DECL PDAT PPDAT128={VEL 100.0,ACC 100.0,APO_DIST 100.0}
DECL PDAT PPDAT129={VEL 100.0,ACC 100.0,APO_DIST 100.0}
DECL E6POS XP110={X 1060.77795,Y 818.632629,Z -11.06633,A 7.32065201,B -48.3011818,C -92.2923126,S 2,T 2,E1 5392.10498,E2 0.0,E3 0.0,E4 0.0,E5 0.0,E6 0.0}
DECL FDAT FP110={TOOL_NO 2,BASE_NO 2,IPO_FRAME #BASE,POINT2[] " ",TQ_STATE FALSE}
DECL PDAT PPDAT130={VEL 100.0,ACC 100.0,APO_DIST 100.0,APO_MODE #CDIS}
DECL E6POS XP111={X 1060.797,Y 818.632324,Z -57.9407082,A 6.91802597,B -40.6268883,C -92.0091476,S 2,T 2,E1 5392.104,E2 0.0,E3 0.0,E4 0.0,E5 0.0,E6 0.0}
DECL FDAT FP111={TOOL_NO 2,BASE_NO 2,IPO_FRAME #BASE,POINT2[] " ",TQ_STATE FALSE}
DECL PDAT PPDAT131={VEL 100.0,ACC 100.0,APO_DIST 100.0,APO_MODE #CDIS}
DECL E6POS XP112={X 1003.49298,Y 1211.995,Z -19.2005291,A 6.74847603,B -43.3643494,C -92.4021835,S 2,T 2,E1 5392.104,E2 0.0,E3 0.0,E4 0.0,E5 0.0,E6 0.0}
DECL FDAT FP112={TOOL_NO 2,BASE_NO 2,IPO_FRAME #BASE,POINT2[] " ",TQ_STATE FALSE}
DECL PDAT PPDAT132={VEL 100.0,ACC 100.0,APO_DIST 100.0,APO_MODE #CDIS}
DECL E6POS XP114={X 1026.76404,Y 1783.36096,Z -11.4180202,A -122.963898,B -25.8167591,C 57.4100609,S 2,T 2,E1 5026.76709,E2 0.0,E3 0.0,E4 0.0,E5 0.0,E6 0.0}
DECL FDAT FP114={TOOL_NO 2,BASE_NO 2,IPO_FRAME #BASE,POINT2[] " ",TQ_STATE FALSE}
DECL PDAT PPDAT134={VEL 100.0,ACC 100.0,APO_DIST 100.0,APO_MODE #CDIS}
DECL E6POS XP119={X -6195.46484,Y 3635.51196,Z -450.273895,A -158.596603,B 3.86077404,C -4.87853193,S 2,T 43,E1 32.7878494,E2 0.0,E3 0.0,E4 0.0,E5 0.0,E6 0.0}
DECL FDAT FP119={TOOL_NO 2,BASE_NO 2,IPO_FRAME #BASE,POINT2[] " ",TQ_STATE FALSE}
DECL PDAT PPDAT139={VEL 100.0,ACC 100.0,APO_DIST 100.0,APO_MODE #CDIS}
DECL PDAT PPDAT140={VEL 100.0,ACC 100.0,APO_DIST 100.0,APO_MODE #CDIS}
DECL E6POS XP120={X 558.198914,Y -840.542419,Z 1190.95898,A 73.9370117,B 3.71631098,C -5.04456091,S 2,T 42,E1 32.7932091,E2 0.0,E3 0.0,E4 0.0,E5 0.0,E6 0.0}
DECL FDAT FP120={TOOL_NO 2,BASE_NO 0,IPO_FRAME #BASE,POINT2[] " ",TQ_STATE FALSE}
DECL PDAT PPDAT141={VEL 100.0,ACC 100.0,APO_DIST 100.0,APO_MODE #CDIS}
DECL E6POS XP121={X -5.26813698,Y 225.397598,Z 1357.05505,A -91.4384232,B 5.65432501,C -0.0243836995,S 2,T 3,E1 866.892273,E2 0.0,E3 0.0,E4 0.0,E5 0.0,E6 0.0}
DECL FDAT FP121={TOOL_NO 2,BASE_NO 0,IPO_FRAME #BASE,POINT2[] " ",TQ_STATE FALSE}
DECL PDAT PPDAT142={VEL 100.0,ACC 100.0,APO_DIST 100.0}
DECL E6POS XP122={X -6762.21094,Y 2715.22705,Z -286.167999,A -1.43572199,B 5.65468884,C -0.0242798794,S 2,T 3,E1 866.892273,E2 0.0,E3 0.0,E4 0.0,E5 0.0,E6 0.0}
DECL FDAT FP122={TOOL_NO 2,BASE_NO 2,IPO_FRAME #BASE,POINT2[] " ",TQ_STATE FALSE}
DECL PDAT PPDAT143={VEL 100.0,ACC 100.0,APO_DIST 100.0,APO_MODE #CDIS}
DECL E6POS XP123={X -6304.68994,Y 3423.53809,Z -312.228088,A 37.3947105,B 0.75025183,C 10.5158195,S 2,T 3,E1 866.892578,E2 0.0,E3 0.0,E4 0.0,E5 0.0,E6 0.0}
DECL FDAT FP123={TOOL_NO 2,BASE_NO 2,IPO_FRAME #BASE,POINT2[] " ",TQ_STATE FALSE}
DECL PDAT PPDAT144={VEL 100.0,ACC 100.0,APO_DIST 100.0,APO_MODE #CDIS}
DECL E6POS XP124={X -5345.3999,Y 3544.12305,Z -363.516602,A 5.63546085,B -3.36820292,C 7.47960901,S 2,T 11,E1 866.885376,E2 0.0,E3 0.0,E4 0.0,E5 0.0,E6 0.0}
DECL FDAT FP124={TOOL_NO 2,BASE_NO 2,IPO_FRAME #BASE,POINT2[] " ",TQ_STATE FALSE}
DECL PDAT PPDAT145={VEL 100.0,ACC 100.0,APO_DIST 100.0,APO_MODE #CDIS}
DECL E6POS XP125={X -4659.89111,Y 2710.31201,Z -340.069885,A -69.4399414,B -4.68788099,C 11.6254101,S 2,T 2,E1 866.890015,E2 0.0,E3 0.0,E4 0.0,E5 0.0,E6 0.0}
DECL FDAT FP125={TOOL_NO 2,BASE_NO 2,IPO_FRAME #BASE,POINT2[] " ",TQ_STATE FALSE}
DECL PDAT PPDAT146={VEL 100.0,ACC 100.0,APO_DIST 100.0,APO_MODE #CDIS}
DECL E6POS XP126={X -4659.89111,Y 2710.31201,Z -340.069885,A -69.4399414,B -4.68788099,C 11.6254101,S 2,T 2,E1 866.890015,E2 0.0,E3 0.0,E4 0.0,E5 0.0,E6 0.0}
DECL FDAT FP126={TOOL_NO 2,BASE_NO 2,IPO_FRAME #BASE,POINT2[] " ",TQ_STATE FALSE}
DECL PDAT PPDAT147={VEL 100.0,ACC 100.0,APO_DIST 100.0,APO_MODE #CDIS}
DECL E6POS XP127={X -5345.3999,Y 3544.12305,Z -363.516602,A 5.63546085,B -3.36820292,C 7.47960901,S 2,T 11,E1 866.885376,E2 0.0,E3 0.0,E4 0.0,E5 0.0,E6 0.0}
DECL FDAT FP127={TOOL_NO 2,BASE_NO 2,IPO_FRAME #BASE,POINT2[] " ",TQ_STATE FALSE}
DECL PDAT PPDAT148={VEL 100.0,ACC 100.0,APO_DIST 100.0,APO_MODE #CDIS}
DECL E6POS XP128={X -6304.68994,Y 3423.53809,Z -312.228088,A 37.3947105,B 0.75025183,C 10.5158195,S 2,T 3,E1 866.892578,E2 0.0,E3 0.0,E4 0.0,E5 0.0,E6 0.0}
DECL FDAT FP128={TOOL_NO 2,BASE_NO 2,IPO_FRAME #BASE,POINT2[] " ",TQ_STATE FALSE}
ENDDAT
